# EPICS substitutions: viocs/si_ps/si_psApp/Db/sfp1.substitutions
file "db/individual.db" {
    pattern { family, pos, num }
        { "SFP1", "02C4", "" }
        { "SFP1", "03C1", "" }
        { "SFP1", "06C4", "" }
        { "SFP1", "07C1", "" }
        { "SFP1", "12C4", "" }
        { "SFP1", "11C1", "" }
        { "SFP1", "14C4", "" }
        { "SFP1", "15C1", "" }
        { "SFP1", "18C4", "" }
        { "SFP1", "19C1", "" }
}
